Module2002.Output.SkillOutput.SkillOutput14.ParameterOutput.ParameterOutput1 := Module[2].Output.SkillOutput[14].ParameterOutput[1];
Module[2].Input.SkillInput[14].ParameterInput[2] := Module2002.Input.SkillInput.SkillInput14.ParameterInput.ParameterInput2;
Module2002.Output.SkillOutput.SkillOutput14.ParameterOutput.ParameterOutput2 := Module[2].Output.SkillOutput[14].ParameterOutput[2];
Module[2].Input.SkillInput[14].ParameterInput[3] := Module2002.Input.SkillInput.SkillInput14.ParameterInput.ParameterInput3;
Module2002.Output.SkillOutput.SkillOutput14.ParameterOutput.ParameterOutput3 := Module[2].Output.SkillOutput[14].ParameterOutput[3];
Module[2].Input.SkillInput[14].ParameterInput[4] := Module2002.Input.SkillInput.SkillInput14.ParameterInput.ParameterInput4;
Module2002.Output.SkillOutput.SkillOutput14.ParameterOutput.ParameterOutput4 := Module[2].Output.SkillOutput[14].ParameterOutput[4];
Module[2].Input.SkillInput[14].ParameterInput[5] := Module2002.Input.SkillInput.SkillInput14.ParameterInput.ParameterInput5;
Module2002.Output.SkillOutput.SkillOutput14.ParameterOutput.ParameterOutput5 := Module[2].Output.SkillOutput[14].ParameterOutput[5];
Module[2].Input.SkillInput[15].Execute := Module2002.Input.SkillInput.SkillInput15.Execute;
Module2002.Output.SkillOutput.SkillOutput15.Dummy := Module[2].Output.SkillOutput[15].Dummy;
Module2002.Output.SkillOutput.SkillOutput15.ID := Module[2].Output.SkillOutput[15].ID;
Module2002.Output.SkillOutput.SkillOutput15.Name := Module[2].Output.SkillOutput[15].Name;
Module2002.Output.SkillOutput.SkillOutput15.Activated := Module[2].Output.SkillOutput[15].Activated;
Module2002.Output.SkillOutput.SkillOutput15.Ready := Module[2].Output.SkillOutput[15].Ready;
Module2002.Output.SkillOutput.SkillOutput15.Busy := Module[2].Output.SkillOutput[15].Busy;
Module2002.Output.SkillOutput.SkillOutput15.Done := Module[2].Output.SkillOutput[15].Done;
Module2002.Output.SkillOutput.SkillOutput15.Error := Module[2].Output.SkillOutput[15].Error;
Module2002.Output.Statevalue.Statevalue0 := Module[2].Output.Statevalue[0];
Module2002.Output.Statevalue.Statevalue1 := Module[2].Output.Statevalue[1];
Module2002.Output.Statevalue.Statevalue2 := Module[2].Output.Statevalue[2];
Module2002.Output.Statevalue.Statevalue3 := Module[2].Output.Statevalue[3];
Module2002.Output.Statevalue.Statevalue4 := Module[2].Output.Statevalue[4];
Module2002.Output.Statevalue.Statevalue5 := Module[2].Output.Statevalue[5];
Module2002.Output.Statevalue.Statevalue6 := Module[2].Output.Statevalue[6];
Module2002.Output.Statevalue.Statevalue7 := Module[2].Output.Statevalue[7];
Module2002.Output.Statevalue.Statevalue8 := Module[2].Output.Statevalue[8];
Module2002.Output.Statevalue.Statevalue9 := Module[2].Output.Statevalue[9];
Module2002.Output.Statevalue.Statevalue10 := Module[2].Output.Statevalue[10];
Module[2].Input.SkillInput[15].ParameterInput[0] := Module2002.Input.SkillInput.SkillInput15.ParameterInput.ParameterInput0;
Module2002.Output.SkillOutput.SkillOutput15.ParameterOutput.ParameterOutput0 := Module[2].Output.SkillOutput[15].ParameterOutput[0];
Module[2].Input.SkillInput[15].ParameterInput[1] := Module2002.Input.SkillInput.SkillInput15.ParameterInput.ParameterInput1;
Module2002.Output.SkillOutput.SkillOutput15.ParameterOutput.ParameterOutput1 := Module[2].Output.SkillOutput[15].ParameterOutput[1];
Module[2].Input.SkillInput[15].ParameterInput[2] := Module2002.Input.SkillInput.SkillInput15.ParameterInput.ParameterInput2;
Module2002.Output.SkillOutput.SkillOutput15.ParameterOutput.ParameterOutput2 := Module[2].Output.SkillOutput[15].ParameterOutput[2];
Module[2].Input.SkillInput[15].ParameterInput[3] := Module2002.Input.SkillInput.SkillInput15.ParameterInput.ParameterInput3;
Module2002.Output.SkillOutput.SkillOutput15.ParameterOutput.ParameterOutput3 := Module[2].Output.SkillOutput[15].ParameterOutput[3];
Module[2].Input.SkillInput[15].ParameterInput[4] := Module2002.Input.SkillInput.SkillInput15.ParameterInput.ParameterInput4;
Module2002.Output.SkillOutput.SkillOutput15.ParameterOutput.ParameterOutput4 := Module[2].Output.SkillOutput[15].ParameterOutput[4];
Module[2].Input.SkillInput[15].ParameterInput[5] := Module2002.Input.SkillInput.SkillInput15.ParameterInput.ParameterInput5;
Module2002.Output.SkillOutput.SkillOutput15.ParameterOutput.ParameterOutput5 := Module[2].Output.SkillOutput[15].ParameterOutput[5];
Module[3].Input.Mode := Module2003.Input.Mode;
Module[3].Input.ConnectionTestInput := Module2003.Input.ConnectionTestInput;
Module[3].Input.PositionInput := Module2003.Input.PositionInput;
Module[3].Input.Watchbit := Module2003.Input.Watchbit;
Module[3].Input.EmergencyStop := Module2003.Input.EmergencyStop;
Module2003.Output.Dummy := Module[3].Output.Dummy;
Module2003.Output.Name := Module[3].Output.Name;
Module2003.Output.ID := Module[3].Output.ID;
Module2003.Output.IP := Module[3].Output.IP;
Module2003.Output.Idle := Module[3].Output.Idle;
Module2003.Output.Connected := Module[3].Output.Connected;
Module2003.Output.Error := Module[3].Output.Error;
Module2003.Output.ErrorID := Module[3].Output.ErrorID;
Module2003.Output.ErrorDescription := Module[3].Output.ErrorDescription;
Module2003.Output.CurrentTaskDescription := Module[3].Output.CurrentTaskDescription;
Module2003.Output.PositionSensor := Module[3].Output.PositionSensor;
Module2003.Output.ConnectionTestOutput := Module[3].Output.ConnectionTestOutput;
Module[3].Input.SkillInput[0].Execute := Module2003.Input.SkillInput.SkillInput0.Execute;
Module2003.Output.SkillOutput.SkillOutput0.Dummy := Module[3].Output.SkillOutput[0].Dummy;
Module2003.Output.SkillOutput.SkillOutput0.ID := Module[3].Output.SkillOutput[0].ID;
Module2003.Output.SkillOutput.SkillOutput0.Name := Module[3].Output.SkillOutput[0].Name;
Module2003.Output.SkillOutput.SkillOutput0.Activated := Module[3].Output.SkillOutput[0].Activated;
Module2003.Output.SkillOutput.SkillOutput0.Ready := Module[3].Output.SkillOutput[0].Ready;
Module2003.Output.SkillOutput.SkillOutput0.Busy := Module[3].Output.SkillOutput[0].Busy;
Module2003.Output.SkillOutput.SkillOutput0.Done := Module[3].Output.SkillOutput[0].Done;
Module2003.Output.SkillOutput.SkillOutput0.Error := Module[3].Output.SkillOutput[0].Error;
Module2003.Output.Statevalue.Statevalue0 := Module[3].Output.Statevalue[0];
Module2003.Output.Statevalue.Statevalue1 := Module[3].Output.Statevalue[1];
Module2003.Output.Statevalue.Statevalue2 := Module[3].Output.Statevalue[2];
Module2003.Output.Statevalue.Statevalue3 := Module[3].Output.Statevalue[3];
Module2003.Output.Statevalue.Statevalue4 := Module[3].Output.Statevalue[4];
Module2003.Output.Statevalue.Statevalue5 := Module[3].Output.Statevalue[5];
Module2003.Output.Statevalue.Statevalue6 := Module[3].Output.Statevalue[6];
Module2003.Output.Statevalue.Statevalue7 := Module[3].Output.Statevalue[7];
Module2003.Output.Statevalue.Statevalue8 := Module[3].Output.Statevalue[8];
Module2003.Output.Statevalue.Statevalue9 := Module[3].Output.Statevalue[9];
Module2003.Output.Statevalue.Statevalue10 := Module[3].Output.Statevalue[10];
Module[3].Input.SkillInput[0].ParameterInput[0] := Module2003.Input.SkillInput.SkillInput0.ParameterInput.ParameterInput0;
Module2003.Output.SkillOutput.SkillOutput0.ParameterOutput.ParameterOutput0 := Module[3].Output.SkillOutput[0].ParameterOutput[0];
Module[3].Input.SkillInput[0].ParameterInput[1] := Module2003.Input.SkillInput.SkillInput0.ParameterInput.ParameterInput1;
Module2003.Output.SkillOutput.SkillOutput0.ParameterOutput.ParameterOutput1 := Module[3].Output.SkillOutput[0].ParameterOutput[1];
Module[3].Input.SkillInput[0].ParameterInput[2] := Module2003.Input.SkillInput.SkillInput0.ParameterInput.ParameterInput2;
Module2003.Output.SkillOutput.SkillOutput0.ParameterOutput.ParameterOutput2 := Module[3].Output.SkillOutput[0].ParameterOutput[2];
Module[3].Input.SkillInput[0].ParameterInput[3] := Module2003.Input.SkillInput.SkillInput0.ParameterInput.ParameterInput3;
Module2003.Output.SkillOutput.SkillOutput0.ParameterOutput.ParameterOutput3 := Module[3].Output.SkillOutput[0].ParameterOutput[3];
Module[3].Input.SkillInput[0].ParameterInput[4] := Module2003.Input.SkillInput.SkillInput0.ParameterInput.ParameterInput4;
Module2003.Output.SkillOutput.SkillOutput0.ParameterOutput.ParameterOutput4 := Module[3].Output.SkillOutput[0].ParameterOutput[4];
Module[3].Input.SkillInput[0].ParameterInput[5] := Module2003.Input.SkillInput.SkillInput0.ParameterInput.ParameterInput5;
Module2003.Output.SkillOutput.SkillOutput0.ParameterOutput.ParameterOutput5 := Module[3].Output.SkillOutput[0].ParameterOutput[5];
Module[3].Input.SkillInput[1].Execute := Module2003.Input.SkillInput.SkillInput1.Execute;
Module2003.Output.SkillOutput.SkillOutput1.Dummy := Module[3].Output.SkillOutput[1].Dummy;
Module2003.Output.SkillOutput.SkillOutput1.ID := Module[3].Output.SkillOutput[1].ID;
Module2003.Output.SkillOutput.SkillOutput1.Name := Module[3].Output.SkillOutput[1].Name;
Module2003.Output.SkillOutput.SkillOutput1.Activated := Module[3].Output.SkillOutput[1].Activated;
Module2003.Output.SkillOutput.SkillOutput1.Ready := Module[3].Output.SkillOutput[1].Ready;
Module2003.Output.SkillOutput.SkillOutput1.Busy := Module[3].Output.SkillOutput[1].Busy;
Module2003.Output.SkillOutput.SkillOutput1.Done := Module[3].Output.SkillOutput[1].Done;
Module2003.Output.SkillOutput.SkillOutput1.Error := Module[3].Output.SkillOutput[1].Error;
Module2003.Output.Statevalue.Statevalue0 := Module[3].Output.Statevalue[0];
Module2003.Output.Statevalue.Statevalue1 := Module[3].Output.Statevalue[1];
Module2003.Output.Statevalue.Statevalue2 := Module[3].Output.Statevalue[2];
Module2003.Output.Statevalue.Statevalue3 := Module[3].Output.Statevalue[3];
Module2003.Output.Statevalue.Statevalue4 := Module[3].Output.Statevalue[4];
Module2003.Output.Statevalue.Statevalue5 := Module[3].Output.Statevalue[5];
Module2003.Output.Statevalue.Statevalue6 := Module[3].Output.Statevalue[6];
Module2003.Output.Statevalue.Statevalue7 := Module[3].Output.Statevalue[7];
Module2003.Output.Statevalue.Statevalue8 := Module[3].Output.Statevalue[8];
Module2003.Output.Statevalue.Statevalue9 := Module[3].Output.Statevalue[9];
Module2003.Output.Statevalue.Statevalue10 := Module[3].Output.Statevalue[10];
Module[3].Input.SkillInput[1].ParameterInput[0] := Module2003.Input.SkillInput.SkillInput1.ParameterInput.ParameterInput0;
Module2003.Output.SkillOutput.SkillOutput1.ParameterOutput.ParameterOutput0 := Module[3].Output.SkillOutput[1].ParameterOutput[0];
Module[3].Input.SkillInput[1].ParameterInput[1] := Module2003.Input.SkillInput.SkillInput1.ParameterInput.ParameterInput1;
Module2003.Output.SkillOutput.SkillOutput1.ParameterOutput.ParameterOutput1 := Module[3].Output.SkillOutput[1].ParameterOutput[1];
Module[3].Input.SkillInput[1].ParameterInput[2] := Module2003.Input.SkillInput.SkillInput1.ParameterInput.ParameterInput2;
Module2003.Output.SkillOutput.SkillOutput1.ParameterOutput.ParameterOutput2 := Module[3].Output.SkillOutput[1].ParameterOutput[2];
Module[3].Input.SkillInput[1].ParameterInput[3] := Module2003.Input.SkillInput.SkillInput1.ParameterInput.ParameterInput3;
Module2003.Output.SkillOutput.SkillOutput1.ParameterOutput.ParameterOutput3 := Module[3].Output.SkillOutput[1].ParameterOutput[3];
Module[3].Input.SkillInput[1].ParameterInput[4] := Module2003.Input.SkillInput.SkillInput1.ParameterInput.ParameterInput4;
Module2003.Output.SkillOutput.SkillOutput1.ParameterOutput.ParameterOutput4 := Module[3].Output.SkillOutput[1].ParameterOutput[4];
Module[3].Input.SkillInput[1].ParameterInput[5] := Module2003.Input.SkillInput.SkillInput1.ParameterInput.ParameterInput5;
Module2003.Output.SkillOutput.SkillOutput1.ParameterOutput.ParameterOutput5 := Module[3].Output.SkillOutput[1].ParameterOutput[5];
Module[3].Input.SkillInput[2].Execute := Module2003.Input.SkillInput.SkillInput2.Execute;
Module2003.Output.SkillOutput.SkillOutput2.Dummy := Module[3].Output.SkillOutput[2].Dummy;
Module2003.Output.SkillOutput.SkillOutput2.ID := Module[3].Output.SkillOutput[2].ID;
Module2003.Output.SkillOutput.SkillOutput2.Name := Module[3].Output.SkillOutput[2].Name;
Module2003.Output.SkillOutput.SkillOutput2.Activated := Module[3].Output.SkillOutput[2].Activated;
Module2003.Output.SkillOutput.SkillOutput2.Ready := Module[3].Output.SkillOutput[2].Ready;
Module2003.Output.SkillOutput.SkillOutput2.Busy := Module[3].Output.SkillOutput[2].Busy;
Module2003.Output.SkillOutput.SkillOutput2.Done := Module[3].Output.SkillOutput[2].Done;
Module2003.Output.SkillOutput.SkillOutput2.Error := Module[3].Output.SkillOutput[2].Error;
Module2003.Output.Statevalue.Statevalue0 := Module[3].Output.Statevalue[0];
Module2003.Output.Statevalue.Statevalue1 := Module[3].Output.Statevalue[1];
Module2003.Output.Statevalue.Statevalue2 := Module[3].Output.Statevalue[2];
Module2003.Output.Statevalue.Statevalue3 := Module[3].Output.Statevalue[3];
Module2003.Output.Statevalue.Statevalue4 := Module[3].Output.Statevalue[4];
Module2003.Output.Statevalue.Statevalue5 := Module[3].Output.Statevalue[5];
Module2003.Output.Statevalue.Statevalue6 := Module[3].Output.Statevalue[6];
Module2003.Output.Statevalue.Statevalue7 := Module[3].Output.Statevalue[7];
Module2003.Output.Statevalue.Statevalue8 := Module[3].Output.Statevalue[8];
Module2003.Output.Statevalue.Statevalue9 := Module[3].Output.Statevalue[9];
Module2003.Output.Statevalue.Statevalue10 := Module[3].Output.Statevalue[10];
Module[3].Input.SkillInput[2].ParameterInput[0] := Module2003.Input.SkillInput.SkillInput2.ParameterInput.ParameterInput0;
Module2003.Output.SkillOutput.SkillOutput2.ParameterOutput.ParameterOutput0 := Module[3].Output.SkillOutput[2].ParameterOutput[0];
Module[3].Input.SkillInput[2].ParameterInput[1] := Module2003.Input.SkillInput.SkillInput2.ParameterInput.ParameterInput1;
Module2003.Output.SkillOutput.SkillOutput2.ParameterOutput.ParameterOutput1 := Module[3].Output.SkillOutput[2].ParameterOutput[1];
Module[3].Input.SkillInput[2].ParameterInput[2] := Module2003.Input.SkillInput.SkillInput2.ParameterInput.ParameterInput2;
Module2003.Output.SkillOutput.SkillOutput2.ParameterOutput.ParameterOutput2 := Module[3].Output.SkillOutput[2].ParameterOutput[2];
Module[3].Input.SkillInput[2].ParameterInput[3] := Module2003.Input.SkillInput.SkillInput2.ParameterInput.ParameterInput3;
Module2003.Output.SkillOutput.SkillOutput2.ParameterOutput.ParameterOutput3 := Module[3].Output.SkillOutput[2].ParameterOutput[3];
Module[3].Input.SkillInput[2].ParameterInput[4] := Module2003.Input.SkillInput.SkillInput2.ParameterInput.ParameterInput4;
Module2003.Output.SkillOutput.SkillOutput2.ParameterOutput.ParameterOutput4 := Module[3].Output.SkillOutput[2].ParameterOutput[4];
Module[3].Input.SkillInput[2].ParameterInput[5] := Module2003.Input.SkillInput.SkillInput2.ParameterInput.ParameterInput5;
Module2003.Output.SkillOutput.SkillOutput2.ParameterOutput.ParameterOutput5 := Module[3].Output.SkillOutput[2].ParameterOutput[5];
Module[3].Input.SkillInput[3].Execute := Module2003.Input.SkillInput.SkillInput3.Execute;
Module2003.Output.SkillOutput.SkillOutput3.Dummy := Module[3].Output.SkillOutput[3].Dummy;
Module2003.Output.SkillOutput.SkillOutput3.ID := Module[3].Output.SkillOutput[3].ID;
Module2003.Output.SkillOutput.SkillOutput3.Name := Module[3].Output.SkillOutput[3].Name;
Module2003.Output.SkillOutput.SkillOutput3.Activated := Module[3].Output.SkillOutput[3].Activated;
Module2003.Output.SkillOutput.SkillOutput3.Ready := Module[3].Output.SkillOutput[3].Ready;
Module2003.Output.SkillOutput.SkillOutput3.Busy := Module[3].Output.SkillOutput[3].Busy;
Module2003.Output.SkillOutput.SkillOutput3.Done := Module[3].Output.SkillOutput[3].Done;
Module2003.Output.SkillOutput.SkillOutput3.Error := Module[3].Output.SkillOutput[3].Error;
Module2003.Output.Statevalue.Statevalue0 := Module[3].Output.Statevalue[0];
Module2003.Output.Statevalue.Statevalue1 := Module[3].Output.Statevalue[1];
Module2003.Output.Statevalue.Statevalue2 := Module[3].Output.Statevalue[2];
Module2003.Output.Statevalue.Statevalue3 := Module[3].Output.Statevalue[3];
Module2003.Output.Statevalue.Statevalue4 := Module[3].Output.Statevalue[4];
Module2003.Output.Statevalue.Statevalue5 := Module[3].Output.Statevalue[5];
Module2003.Output.Statevalue.Statevalue6 := Module[3].Output.Statevalue[6];
Module2003.Output.Statevalue.Statevalue7 := Module[3].Output.Statevalue[7];
Module2003.Output.Statevalue.Statevalue8 := Module[3].Output.Statevalue[8];
Module2003.Output.Statevalue.Statevalue9 := Module[3].Output.Statevalue[9];
Module2003.Output.Statevalue.Statevalue10 := Module[3].Output.Statevalue[10];
Module[3].Input.SkillInput[3].ParameterInput[0] := Module2003.Input.SkillInput.SkillInput3.ParameterInput.ParameterInput0;
Module2003.Output.SkillOutput.SkillOutput3.ParameterOutput.ParameterOutput0 := Module[3].Output.SkillOutput[3].ParameterOutput[0];
Module[3].Input.SkillInput[3].ParameterInput[1] := Module2003.Input.SkillInput.SkillInput3.ParameterInput.ParameterInput1;
Module2003.Output.SkillOutput.SkillOutput3.ParameterOutput.ParameterOutput1 := Module[3].Output.SkillOutput[3].ParameterOutput[1];
Module[3].Input.SkillInput[3].ParameterInput[2] := Module2003.Input.SkillInput.SkillInput3.ParameterInput.ParameterInput2;
Module2003.Output.SkillOutput.SkillOutput3.ParameterOutput.ParameterOutput2 := Module[3].Output.SkillOutput[3].ParameterOutput[2];
Module[3].Input.SkillInput[3].ParameterInput[3] := Module2003.Input.SkillInput.SkillInput3.ParameterInput.ParameterInput3;
Module2003.Output.SkillOutput.SkillOutput3.ParameterOutput.ParameterOutput3 := Module[3].Output.SkillOutput[3].ParameterOutput[3];
Module[3].Input.SkillInput[3].ParameterInput[4] := Module2003.Input.SkillInput.SkillInput3.ParameterInput.ParameterInput4;
Module2003.Output.SkillOutput.SkillOutput3.ParameterOutput.ParameterOutput4 := Module[3].Output.SkillOutput[3].ParameterOutput[4];
Module[3].Input.SkillInput[3].ParameterInput[5] := Module2003.Input.SkillInput.SkillInput3.ParameterInput.ParameterInput5;
Module2003.Output.SkillOutput.SkillOutput3.ParameterOutput.ParameterOutput5 := Module[3].Output.SkillOutput[3].ParameterOutput[5];
Module[3].Input.SkillInput[4].Execute := Module2003.Input.SkillInput.SkillInput4.Execute;
Module2003.Output.SkillOutput.SkillOutput4.Dummy := Module[3].Output.SkillOutput[4].Dummy;
Module2003.Output.SkillOutput.SkillOutput4.ID := Module[3].Output.SkillOutput[4].ID;
Module2003.Output.SkillOutput.SkillOutput4.Name := Module[3].Output.SkillOutput[4].Name;
Module2003.Output.SkillOutput.SkillOutput4.Activated := Module[3].Output.SkillOutput[4].Activated;
Module2003.Output.SkillOutput.SkillOutput4.Ready := Module[3].Output.SkillOutput[4].Ready;
Module2003.Output.SkillOutput.SkillOutput4.Busy := Module[3].Output.SkillOutput[4].Busy;
Module2003.Output.SkillOutput.SkillOutput4.Done := Module[3].Output.SkillOutput[4].Done;
Module2003.Output.SkillOutput.SkillOutput4.Error := Module[3].Output.SkillOutput[4].Error;
Module2003.Output.Statevalue.Statevalue0 := Module[3].Output.Statevalue[0];
Module2003.Output.Statevalue.Statevalue1 := Module[3].Output.Statevalue[1];
Module2003.Output.Statevalue.Statevalue2 := Module[3].Output.Statevalue[2];
Module2003.Output.Statevalue.Statevalue3 := Module[3].Output.Statevalue[3];
Module2003.Output.Statevalue.Statevalue4 := Module[3].Output.Statevalue[4];
Module2003.Output.Statevalue.Statevalue5 := Module[3].Output.Statevalue[5];
Module2003.Output.Statevalue.Statevalue6 := Module[3].Output.Statevalue[6];
Module2003.Output.Statevalue.Statevalue7 := Module[3].Output.Statevalue[7];
Module2003.Output.Statevalue.Statevalue8 := Module[3].Output.Statevalue[8];
Module2003.Output.Statevalue.Statevalue9 := Module[3].Output.Statevalue[9];
Module2003.Output.Statevalue.Statevalue10 := Module[3].Output.Statevalue[10];
Module[3].Input.SkillInput[4].ParameterInput[0] := Module2003.Input.SkillInput.SkillInput4.ParameterInput.ParameterInput0;
Module2003.Output.SkillOutput.SkillOutput4.ParameterOutput.ParameterOutput0 := Module[3].Output.SkillOutput[4].ParameterOutput[0];
Module[3].Input.SkillInput[4].ParameterInput[1] := Module2003.Input.SkillInput.SkillInput4.ParameterInput.ParameterInput1;
Module2003.Output.SkillOutput.SkillOutput4.ParameterOutput.ParameterOutput1 := Module[3].Output.SkillOutput[4].ParameterOutput[1];
Module[3].Input.SkillInput[4].ParameterInput[2] := Module2003.Input.SkillInput.SkillInput4.ParameterInput.ParameterInput2;
Module2003.Output.SkillOutput.SkillOutput4.ParameterOutput.ParameterOutput2 := Module[3].Output.SkillOutput[4].ParameterOutput[2];
Module[3].Input.SkillInput[4].ParameterInput[3] := Module2003.Input.SkillInput.SkillInput4.ParameterInput.ParameterInput3;
Module2003.Output.SkillOutput.SkillOutput4.ParameterOutput.ParameterOutput3 := Module[3].Output.SkillOutput[4].ParameterOutput[3];
Module[3].Input.SkillInput[4].ParameterInput[4] := Module2003.Input.SkillInput.SkillInput4.ParameterInput.ParameterInput4;
Module2003.Output.SkillOutput.SkillOutput4.ParameterOutput.ParameterOutput4 := Module[3].Output.SkillOutput[4].ParameterOutput[4];
Module[3].Input.SkillInput[4].ParameterInput[5] := Module2003.Input.SkillInput.SkillInput4.ParameterInput.ParameterInput5;
Module2003.Output.SkillOutput.SkillOutput4.ParameterOutput.ParameterOutput5 := Module[3].Output.SkillOutput[4].ParameterOutput[5];
Module[3].Input.SkillInput[5].Execute := Module2003.Input.SkillInput.SkillInput5.Execute;
Module2003.Output.SkillOutput.SkillOutput5.Dummy := Module[3].Output.SkillOutput[5].Dummy;
Module2003.Output.SkillOutput.SkillOutput5.ID := Module[3].Output.SkillOutput[5].ID;
Module2003.Output.SkillOutput.SkillOutput5.Name := Module[3].Output.SkillOutput[5].Name;
Module2003.Output.SkillOutput.SkillOutput5.Activated := Module[3].Output.SkillOutput[5].Activated;
Module2003.Output.SkillOutput.SkillOutput5.Ready := Module[3].Output.SkillOutput[5].Ready;
Module2003.Output.SkillOutput.SkillOutput5.Busy := Module[3].Output.SkillOutput[5].Busy;
Module2003.Output.SkillOutput.SkillOutput5.Done := Module[3].Output.SkillOutput[5].Done;
Module2003.Output.SkillOutput.SkillOutput5.Error := Module[3].Output.SkillOutput[5].Error;
Module2003.Output.Statevalue.Statevalue0 := Module[3].Output.Statevalue[0];
Module2003.Output.Statevalue.Statevalue1 := Module[3].Output.Statevalue[1];
Module2003.Output.Statevalue.Statevalue2 := Module[3].Output.Statevalue[2];
Module2003.Output.Statevalue.Statevalue3 := Module[3].Output.Statevalue[3];
Module2003.Output.Statevalue.Statevalue4 := Module[3].Output.Statevalue[4];
Module2003.Output.Statevalue.Statevalue5 := Module[3].Output.Statevalue[5];
Module2003.Output.Statevalue.Statevalue6 := Module[3].Output.Statevalue[6];
Module2003.Output.Statevalue.Statevalue7 := Module[3].Output.Statevalue[7];
Module2003.Output.Statevalue.Statevalue8 := Module[3].Output.Statevalue[8];
Module2003.Output.Statevalue.Statevalue9 := Module[3].Output.Statevalue[9];
Module2003.Output.Statevalue.Statevalue10 := Module[3].Output.Statevalue[10];
Module[3].Input.SkillInput[5].ParameterInput[0] := Module2003.Input.SkillInput.SkillInput5.ParameterInput.ParameterInput0;
Module2003.Output.SkillOutput.SkillOutput5.ParameterOutput.ParameterOutput0 := Module[3].Output.SkillOutput[5].ParameterOutput[0];
Module[3].Input.SkillInput[5].ParameterInput[1] := Module2003.Input.SkillInput.SkillInput5.ParameterInput.ParameterInput1;
Module2003.Output.SkillOutput.SkillOutput5.ParameterOutput.ParameterOutput1 := Module[3].Output.SkillOutput[5].ParameterOutput[1];
Module[3].Input.SkillInput[5].ParameterInput[2] := Module2003.Input.SkillInput.SkillInput5.ParameterInput.ParameterInput2;
Module2003.Output.SkillOutput.SkillOutput5.ParameterOutput.ParameterOutput2 := Module[3].Output.SkillOutput[5].ParameterOutput[2];
Module[3].Input.SkillInput[5].ParameterInput[3] := Module2003.Input.SkillInput.SkillInput5.ParameterInput.ParameterInput3;
Module2003.Output.SkillOutput.SkillOutput5.ParameterOutput.ParameterOutput3 := Module[3].Output.SkillOutput[5].ParameterOutput[3];
Module[3].Input.SkillInput[5].ParameterInput[4] := Module2003.Input.SkillInput.SkillInput5.ParameterInput.ParameterInput4;
Module2003.Output.SkillOutput.SkillOutput5.ParameterOutput.ParameterOutput4 := Module[3].Output.SkillOutput[5].ParameterOutput[4];
Module[3].Input.SkillInput[5].ParameterInput[5] := Module2003.Input.SkillInput.SkillInput5.ParameterInput.ParameterInput5;
Module2003.Output.SkillOutput.SkillOutput5.ParameterOutput.ParameterOutput5 := Module[3].Output.SkillOutput[5].ParameterOutput[5];
Module[3].Input.SkillInput[6].Execute := Module2003.Input.SkillInput.SkillInput6.Execute;
Module2003.Output.SkillOutput.SkillOutput6.Dummy := Module[3].Output.SkillOutput[6].Dummy;
Module2003.Output.SkillOutput.SkillOutput6.ID := Module[3].Output.SkillOutput[6].ID;
Module2003.Output.SkillOutput.SkillOutput6.Name := Module[3].Output.SkillOutput[6].Name;
Module2003.Output.SkillOutput.SkillOutput6.Activated := Module[3].Output.SkillOutput[6].Activated;
Module2003.Output.SkillOutput.SkillOutput6.Ready := Module[3].Output.SkillOutput[6].Ready;
Module2003.Output.SkillOutput.SkillOutput6.Busy := Module[3].Output.SkillOutput[6].Busy;
Module2003.Output.SkillOutput.SkillOutput6.Done := Module[3].Output.SkillOutput[6].Done;
Module2003.Output.SkillOutput.SkillOutput6.Error := Module[3].Output.SkillOutput[6].Error;
Module2003.Output.Statevalue.Statevalue0 := Module[3].Output.Statevalue[0];
Module2003.Output.Statevalue.Statevalue1 := Module[3].Output.Statevalue[1];
Module2003.Output.Statevalue.Statevalue2 := Module[3].Output.Statevalue[2];
Module2003.Output.Statevalue.Statevalue3 := Module[3].Output.Statevalue[3];
Module2003.Output.Statevalue.Statevalue4 := Module[3].Output.Statevalue[4];
Module2003.Output.Statevalue.Statevalue5 := Module[3].Output.Statevalue[5];
Module2003.Output.Statevalue.Statevalue6 := Module[3].Output.Statevalue[6];
Module2003.Output.Statevalue.Statevalue7 := Module[3].Output.Statevalue[7];
Module2003.Output.Statevalue.Statevalue8 := Module[3].Output.Statevalue[8];
Module2003.Output.Statevalue.Statevalue9 := Module[3].Output.Statevalue[9];
Module2003.Output.Statevalue.Statevalue10 := Module[3].Output.Statevalue[10];
Module[3].Input.SkillInput[6].ParameterInput[0] := Module2003.Input.SkillInput.SkillInput6.ParameterInput.ParameterInput0;
Module2003.Output.SkillOutput.SkillOutput6.ParameterOutput.ParameterOutput0 := Module[3].Output.SkillOutput[6].ParameterOutput[0];
Module[3].Input.SkillInput[6].ParameterInput[1] := Module2003.Input.SkillInput.SkillInput6.ParameterInput.ParameterInput1;
Module2003.Output.SkillOutput.SkillOutput6.ParameterOutput.ParameterOutput1 := Module[3].Output.SkillOutput[6].ParameterOutput[1];
Module[3].Input.SkillInput[6].ParameterInput[2] := Module2003.Input.SkillInput.SkillInput6.ParameterInput.ParameterInput2;
Module2003.Output.SkillOutput.SkillOutput6.ParameterOutput.ParameterOutput2 := Module[3].Output.SkillOutput[6].ParameterOutput[2];
Module[3].Input.SkillInput[6].ParameterInput[3] := Module2003.Input.SkillInput.SkillInput6.ParameterInput.ParameterInput3;
Module2003.Output.SkillOutput.SkillOutput6.ParameterOutput.ParameterOutput3 := Module[3].Output.SkillOutput[6].ParameterOutput[3];
Module[3].Input.SkillInput[6].ParameterInput[4] := Module2003.Input.SkillInput.SkillInput6.ParameterInput.ParameterInput4;
Module2003.Output.SkillOutput.SkillOutput6.ParameterOutput.ParameterOutput4 := Module[3].Output.SkillOutput[6].ParameterOutput[4];
Module[3].Input.SkillInput[6].ParameterInput[5] := Module2003.Input.SkillInput.SkillInput6.ParameterInput.ParameterInput5;
Module2003.Output.SkillOutput.SkillOutput6.ParameterOutput.ParameterOutput5 := Module[3].Output.SkillOutput[6].ParameterOutput[5];
Module[3].Input.SkillInput[7].Execute := Module2003.Input.SkillInput.SkillInput7.Execute;
Module2003.Output.SkillOutput.SkillOutput7.Dummy := Module[3].Output.SkillOutput[7].Dummy;
Module2003.Output.SkillOutput.SkillOutput7.ID := Module[3].Output.SkillOutput[7].ID;
Module2003.Output.SkillOutput.SkillOutput7.Name := Module[3].Output.SkillOutput[7].Name;
Module2003.Output.SkillOutput.SkillOutput7.Activated := Module[3].Output.SkillOutput[7].Activated;
Module2003.Output.SkillOutput.SkillOutput7.Ready := Module[3].Output.SkillOutput[7].Ready;
Module2003.Output.SkillOutput.SkillOutput7.Busy := Module[3].Output.SkillOutput[7].Busy;
Module2003.Output.SkillOutput.SkillOutput7.Done := Module[3].Output.SkillOutput[7].Done;
Module2003.Output.SkillOutput.SkillOutput7.Error := Module[3].Output.SkillOutput[7].Error;
Module2003.Output.Statevalue.Statevalue0 := Module[3].Output.Statevalue[0];
Module2003.Output.Statevalue.Statevalue1 := Module[3].Output.Statevalue[1];
Module2003.Output.Statevalue.Statevalue2 := Module[3].Output.Statevalue[2];
Module2003.Output.Statevalue.Statevalue3 := Module[3].Output.Statevalue[3];
Module2003.Output.Statevalue.Statevalue4 := Module[3].Output.Statevalue[4];
Module2003.Output.Statevalue.Statevalue5 := Module[3].Output.Statevalue[5];
Module2003.Output.Statevalue.Statevalue6 := Module[3].Output.Statevalue[6];
Module2003.Output.Statevalue.Statevalue7 := Module[3].Output.Statevalue[7];
Module2003.Output.Statevalue.Statevalue8 := Module[3].Output.Statevalue[8];
Module2003.Output.Statevalue.Statevalue9 := Module[3].Output.Statevalue[9];
Module2003.Output.Statevalue.Statevalue10 := Module[3].Output.Statevalue[10];
Module[3].Input.SkillInput[7].ParameterInput[0] := Module2003.Input.SkillInput.SkillInput7.ParameterInput.ParameterInput0;
Module2003.Output.SkillOutput.SkillOutput7.ParameterOutput.ParameterOutput0 := Module[3].Output.SkillOutput[7].ParameterOutput[0];
Module[3].Input.SkillInput[7].ParameterInput[1] := Module2003.Input.SkillInput.SkillInput7.ParameterInput.ParameterInput1;
Module2003.Output.SkillOutput.SkillOutput7.ParameterOutput.ParameterOutput1 := Module[3].Output.SkillOutput[7].ParameterOutput[1];
Module[3].Input.SkillInput[7].ParameterInput[2] := Module2003.Input.SkillInput.SkillInput7.ParameterInput.ParameterInput2;
Module2003.Output.SkillOutput.SkillOutput7.ParameterOutput.ParameterOutput2 := Module[3].Output.SkillOutput[7].ParameterOutput[2];
Module[3].Input.SkillInput[7].ParameterInput[3] := Module2003.Input.SkillInput.SkillInput7.ParameterInput.ParameterInput3;
Module2003.Output.SkillOutput.SkillOutput7.ParameterOutput.ParameterOutput3 := Module[3].Output.SkillOutput[7].ParameterOutput[3];
Module[3].Input.SkillInput[7].ParameterInput[4] := Module2003.Input.SkillInput.SkillInput7.ParameterInput.ParameterInput4;
Module2003.Output.SkillOutput.SkillOutput7.ParameterOutput.ParameterOutput4 := Module[3].Output.SkillOutput[7].ParameterOutput[4];
Module[3].Input.SkillInput[7].ParameterInput[5] := Module2003.Input.SkillInput.SkillInput7.ParameterInput.ParameterInput5;
Module2003.Output.SkillOutput.SkillOutput7.ParameterOutput.ParameterOutput5 := Module[3].Output.SkillOutput[7].ParameterOutput[5];
Module[3].Input.SkillInput[8].Execute := Module2003.Input.SkillInput.SkillInput8.Execute;
Module2003.Output.SkillOutput.SkillOutput8.Dummy := Module[3].Output.SkillOutput[8].Dummy;
Module2003.Output.SkillOutput.SkillOutput8.ID := Module[3].Output.SkillOutput[8].ID;
Module2003.Output.SkillOutput.SkillOutput8.Name := Module[3].Output.SkillOutput[8].Name;
Module2003.Output.SkillOutput.SkillOutput8.Activated := Module[3].Output.SkillOutput[8].Activated;
Module2003.Output.SkillOutput.SkillOutput8.Ready := Module[3].Output.SkillOutput[8].Ready;
Module2003.Output.SkillOutput.SkillOutput8.Busy := Module[3].Output.SkillOutput[8].Busy;
Module2003.Output.SkillOutput.SkillOutput8.Done := Module[3].Output.SkillOutput[8].Done;
Module2003.Output.SkillOutput.SkillOutput8.Error := Module[3].Output.SkillOutput[8].Error;
Module2003.Output.Statevalue.Statevalue0 := Module[3].Output.Statevalue[0];
Module2003.Output.Statevalue.Statevalue1 := Module[3].Output.Statevalue[1];
Module2003.Output.Statevalue.Statevalue2 := Module[3].Output.Statevalue[2];
Module2003.Output.Statevalue.Statevalue3 := Module[3].Output.Statevalue[3];
Module2003.Output.Statevalue.Statevalue4 := Module[3].Output.Statevalue[4];
Module2003.Output.Statevalue.Statevalue5 := Module[3].Output.Statevalue[5];
Module2003.Output.Statevalue.Statevalue6 := Module[3].Output.Statevalue[6];
Module2003.Output.Statevalue.Statevalue7 := Module[3].Output.Statevalue[7];
Module2003.Output.Statevalue.Statevalue8 := Module[3].Output.Statevalue[8];
Module2003.Output.Statevalue.Statevalue9 := Module[3].Output.Statevalue[9];
Module2003.Output.Statevalue.Statevalue10 := Module[3].Output.Statevalue[10];
Module[3].Input.SkillInput[8].ParameterInput[0] := Module2003.Input.SkillInput.SkillInput8.ParameterInput.ParameterInput0;
Module2003.Output.SkillOutput.SkillOutput8.ParameterOutput.ParameterOutput0 := Module[3].Output.SkillOutput[8].ParameterOutput[0];
Module[3].Input.SkillInput[8].ParameterInput[1] := Module2003.Input.SkillInput.SkillInput8.ParameterInput.ParameterInput1;
Module2003.Output.SkillOutput.SkillOutput8.ParameterOutput.ParameterOutput1 := Module[3].Output.SkillOutput[8].ParameterOutput[1];
Module[3].Input.SkillInput[8].ParameterInput[2] := Module2003.Input.SkillInput.SkillInput8.ParameterInput.ParameterInput2;
Module2003.Output.SkillOutput.SkillOutput8.ParameterOutput.ParameterOutput2 := Module[3].Output.SkillOutput[8].ParameterOutput[2];
Module[3].Input.SkillInput[8].ParameterInput[3] := Module2003.Input.SkillInput.SkillInput8.ParameterInput.ParameterInput3;
Module2003.Output.SkillOutput.SkillOutput8.ParameterOutput.ParameterOutput3 := Module[3].Output.SkillOutput[8].ParameterOutput[3];
Module[3].Input.SkillInput[8].ParameterInput[4] := Module2003.Input.SkillInput.SkillInput8.ParameterInput.ParameterInput4;
Module2003.Output.SkillOutput.SkillOutput8.ParameterOutput.ParameterOutput4 := Module[3].Output.SkillOutput[8].ParameterOutput[4];
Module[3].Input.SkillInput[8].ParameterInput[5] := Module2003.Input.SkillInput.SkillInput8.ParameterInput.ParameterInput5;
Module2003.Output.SkillOutput.SkillOutput8.ParameterOutput.ParameterOutput5 := Module[3].Output.SkillOutput[8].ParameterOutput[5];
Module[3].Input.SkillInput[9].Execute := Module2003.Input.SkillInput.SkillInput9.Execute;
Module2003.Output.SkillOutput.SkillOutput9.Dummy := Module[3].Output.SkillOutput[9].Dummy;
Module2003.Output.SkillOutput.SkillOutput9.ID := Module[3].Output.SkillOutput[9].ID;
Module2003.Output.SkillOutput.SkillOutput9.Name := Module[3].Output.SkillOutput[9].Name;
Module2003.Output.SkillOutput.SkillOutput9.Activated := Module[3].Output.SkillOutput[9].Activated;
Module2003.Output.SkillOutput.SkillOutput9.Ready := Module[3].Output.SkillOutput[9].Ready;
Module2003.Output.SkillOutput.SkillOutput9.Busy := Module[3].Output.SkillOutput[9].Busy;
Module2003.Output.SkillOutput.SkillOutput9.Done := Module[3].Output.SkillOutput[9].Done;
Module2003.Output.SkillOutput.SkillOutput9.Error := Module[3].Output.SkillOutput[9].Error;
Module2003.Output.Statevalue.Statevalue0 := Module[3].Output.Statevalue[0];
Module2003.Output.Statevalue.Statevalue1 := Module[3].Output.Statevalue[1];
Module2003.Output.Statevalue.Statevalue2 := Module[3].Output.Statevalue[2];
Module2003.Output.Statevalue.Statevalue3 := Module[3].Output.Statevalue[3];
Module2003.Output.Statevalue.Statevalue4 := Module[3].Output.Statevalue[4];
Module2003.Output.Statevalue.Statevalue5 := Module[3].Output.Statevalue[5];
Module2003.Output.Statevalue.Statevalue6 := Module[3].Output.Statevalue[6];
Module2003.Output.Statevalue.Statevalue7 := Module[3].Output.Statevalue[7];
Module2003.Output.Statevalue.Statevalue8 := Module[3].Output.Statevalue[8];
Module2003.Output.Statevalue.Statevalue9 := Module[3].Output.Statevalue[9];
Module2003.Output.Statevalue.Statevalue10 := Module[3].Output.Statevalue[10];
Module[3].Input.SkillInput[9].ParameterInput[0] := Module2003.Input.SkillInput.SkillInput9.ParameterInput.ParameterInput0;
Module2003.Output.SkillOutput.SkillOutput9.ParameterOutput.ParameterOutput0 := Module[3].Output.SkillOutput[9].ParameterOutput[0];
Module[3].Input.SkillInput[9].ParameterInput[1] := Module2003.Input.SkillInput.SkillInput9.ParameterInput.ParameterInput1;
Module2003.Output.SkillOutput.SkillOutput9.ParameterOutput.ParameterOutput1 := Module[3].Output.SkillOutput[9].ParameterOutput[1];
Module[3].Input.SkillInput[9].ParameterInput[2] := Module2003.Input.SkillInput.SkillInput9.ParameterInput.ParameterInput2;
Module2003.Output.SkillOutput.SkillOutput9.ParameterOutput.ParameterOutput2 := Module[3].Output.SkillOutput[9].ParameterOutput[2];
Module[3].Input.SkillInput[9].ParameterInput[3] := Module2003.Input.SkillInput.SkillInput9.ParameterInput.ParameterInput3;
Module2003.Output.SkillOutput.SkillOutput9.ParameterOutput.ParameterOutput3 := Module[3].Output.SkillOutput[9].ParameterOutput[3];
Module[3].Input.SkillInput[9].ParameterInput[4] := Module2003.Input.SkillInput.SkillInput9.ParameterInput.ParameterInput4;
Module2003.Output.SkillOutput.SkillOutput9.ParameterOutput.ParameterOutput4 := Module[3].Output.SkillOutput[9].ParameterOutput[4];
Module[3].Input.SkillInput[9].ParameterInput[5] := Module2003.Input.SkillInput.SkillInput9.ParameterInput.ParameterInput5;
Module2003.Output.SkillOutput.SkillOutput9.ParameterOutput.ParameterOutput5 := Module[3].Output.SkillOutput[9].ParameterOutput[5];
Module[3].Input.SkillInput[10].Execute := Module2003.Input.SkillInput.SkillInput10.Execute;
Module2003.Output.SkillOutput.SkillOutput10.Dummy := Module[3].Output.SkillOutput[10].Dummy;
Module2003.Output.SkillOutput.SkillOutput10.ID := Module[3].Output.SkillOutput[10].ID;
Module2003.Output.SkillOutput.SkillOutput10.Name := Module[3].Output.SkillOutput[10].Name;
Module2003.Output.SkillOutput.SkillOutput10.Activated := Module[3].Output.SkillOutput[10].Activated;
Module2003.Output.SkillOutput.SkillOutput10.Ready := Module[3].Output.SkillOutput[10].Ready;
Module2003.Output.SkillOutput.SkillOutput10.Busy := Module[3].Output.SkillOutput[10].Busy;
Module2003.Output.SkillOutput.SkillOutput10.Done := Module[3].Output.SkillOutput[10].Done;
Module2003.Output.SkillOutput.SkillOutput10.Error := Module[3].Output.SkillOutput[10].Error;
Module2003.Output.Statevalue.Statevalue0 := Module[3].Output.Statevalue[0];
Module2003.Output.Statevalue.Statevalue1 := Module[3].Output.Statevalue[1];
Module2003.Output.Statevalue.Statevalue2 := Module[3].Output.Statevalue[2];
Module2003.Output.Statevalue.Statevalue3 := Module[3].Output.Statevalue[3];
Module2003.Output.Statevalue.Statevalue4 := Module[3].Output.Statevalue[4];
Module2003.Output.Statevalue.Statevalue5 := Module[3].Output.Statevalue[5];
Module2003.Output.Statevalue.Statevalue6 := Module[3].Output.Statevalue[6];
Module2003.Output.Statevalue.Statevalue7 := Module[3].Output.Statevalue[7];
Module2003.Output.Statevalue.Statevalue8 := Module[3].Output.Statevalue[8];
Module2003.Output.Statevalue.Statevalue9 := Module[3].Output.Statevalue[9];
Module2003.Output.Statevalue.Statevalue10 := Module[3].Output.Statevalue[10];
Module[3].Input.SkillInput[10].ParameterInput[0] := Module2003.Input.SkillInput.SkillInput10.ParameterInput.ParameterInput0;
Module2003.Output.SkillOutput.SkillOutput10.ParameterOutput.ParameterOutput0 := Module[3].Output.SkillOutput[10].ParameterOutput[0];
Module[3].Input.SkillInput[10].ParameterInput[1] := Module2003.Input.SkillInput.SkillInput10.ParameterInput.ParameterInput1;
Module2003.Output.SkillOutput.SkillOutput10.ParameterOutput.ParameterOutput1 := Module[3].Output.SkillOutput[10].ParameterOutput[1];
Module[3].Input.SkillInput[10].ParameterInput[2] := Module2003.Input.SkillInput.SkillInput10.ParameterInput.ParameterInput2;
Module2003.Output.SkillOutput.SkillOutput10.ParameterOutput.ParameterOutput2 := Module[3].Output.SkillOutput[10].ParameterOutput[2];
Module[3].Input.SkillInput[10].ParameterInput[3] := Module2003.Input.SkillInput.SkillInput10.ParameterInput.ParameterInput3;
Module2003.Output.SkillOutput.SkillOutput10.ParameterOutput.ParameterOutput3 := Module[3].Output.SkillOutput[10].ParameterOutput[3];
Module[3].Input.SkillInput[10].ParameterInput[4] := Module2003.Input.SkillInput.SkillInput10.ParameterInput.ParameterInput4;
Module2003.Output.SkillOutput.SkillOutput10.ParameterOutput.ParameterOutput4 := Module[3].Output.SkillOutput[10].ParameterOutput[4];
Module[3].Input.SkillInput[10].ParameterInput[5] := Module2003.Input.SkillInput.SkillInput10.ParameterInput.ParameterInput5;
Module2003.Output.SkillOutput.SkillOutput10.ParameterOutput.ParameterOutput5 := Module[3].Output.SkillOutput[10].ParameterOutput[5];
Module[3].Input.SkillInput[11].Execute := Module2003.Input.SkillInput.SkillInput11.Execute;
Module2003.Output.SkillOutput.SkillOutput11.Dummy := Module[3].Output.SkillOutput[11].Dummy;
Module2003.Output.SkillOutput.SkillOutput11.ID := Module[3].Output.SkillOutput[11].ID;
Module2003.Output.SkillOutput.SkillOutput11.Name := Module[3].Output.SkillOutput[11].Name;
Module2003.Output.SkillOutput.SkillOutput11.Activated := Module[3].Output.SkillOutput[11].Activated;
Module2003.Output.SkillOutput.SkillOutput11.Ready := Module[3].Output.SkillOutput[11].Ready;
Module2003.Output.SkillOutput.SkillOutput11.Busy := Module[3].Output.SkillOutput[11].Busy;
Module2003.Output.SkillOutput.SkillOutput11.Done := Module[3].Output.SkillOutput[11].Done;
Module2003.Output.SkillOutput.SkillOutput11.Error := Module[3].Output.SkillOutput[11].Error;
Module2003.Output.Statevalue.Statevalue0 := Module[3].Output.Statevalue[0];
Module2003.Output.Statevalue.Statevalue1 := Module[3].Output.Statevalue[1];
Module2003.Output.Statevalue.Statevalue2 := Module[3].Output.Statevalue[2];
Module2003.Output.Statevalue.Statevalue3 := Module[3].Output.Statevalue[3];
Module2003.Output.Statevalue.Statevalue4 := Module[3].Output.Statevalue[4];
Module2003.Output.Statevalue.Statevalue5 := Module[3].Output.Statevalue[5];
Module2003.Output.Statevalue.Statevalue6 := Module[3].Output.Statevalue[6];
Module2003.Output.Statevalue.Statevalue7 := Module[3].Output.Statevalue[7];
Module2003.Output.Statevalue.Statevalue8 := Module[3].Output.Statevalue[8];
Module2003.Output.Statevalue.Statevalue9 := Module[3].Output.Statevalue[9];
Module2003.Output.Statevalue.Statevalue10 := Module[3].Output.Statevalue[10];
Module[3].Input.SkillInput[11].ParameterInput[0] := Module2003.Input.SkillInput.SkillInput11.ParameterInput.ParameterInput0;
Module2003.Output.SkillOutput.SkillOutput11.ParameterOutput.ParameterOutput0 := Module[3].Output.SkillOutput[11].ParameterOutput[0];
Module[3].Input.SkillInput[11].ParameterInput[1] := Module2003.Input.SkillInput.SkillInput11.ParameterInput.ParameterInput1;
Module2003.Output.SkillOutput.SkillOutput11.ParameterOutput.ParameterOutput1 := Module[3].Output.SkillOutput[11].ParameterOutput[1];
Module[3].Input.SkillInput[11].ParameterInput[2] := Module2003.Input.SkillInput.SkillInput11.ParameterInput.ParameterInput2;
Module2003.Output.SkillOutput.SkillOutput11.ParameterOutput.ParameterOutput2 := Module[3].Output.SkillOutput[11].ParameterOutput[2];
Module[3].Input.SkillInput[11].ParameterInput[3] := Module2003.Input.SkillInput.SkillInput11.ParameterInput.ParameterInput3;
Module2003.Output.SkillOutput.SkillOutput11.ParameterOutput.ParameterOutput3 := Module[3].Output.SkillOutput[11].ParameterOutput[3];
Module[3].Input.SkillInput[11].ParameterInput[4] := Module2003.Input.SkillInput.SkillInput11.ParameterInput.ParameterInput4;
Module2003.Output.SkillOutput.SkillOutput11.ParameterOutput.ParameterOutput4 := Module[3].Output.SkillOutput[11].ParameterOutput[4];
Module[3].Input.SkillInput[11].ParameterInput[5] := Module2003.Input.SkillInput.SkillInput11.ParameterInput.ParameterInput5;
Module2003.Output.SkillOutput.SkillOutput11.ParameterOutput.ParameterOutput5 := Module[3].Output.SkillOutput[11].ParameterOutput[5];
Module[3].Input.SkillInput[12].Execute := Module2003.Input.SkillInput.SkillInput12.Execute;
Module2003.Output.SkillOutput.SkillOutput12.Dummy := Module[3].Output.SkillOutput[12].Dummy;
Module2003.Output.SkillOutput.SkillOutput12.ID := Module[3].Output.SkillOutput[12].ID;
Module2003.Output.SkillOutput.SkillOutput12.Name := Module[3].Output.SkillOutput[12].Name;
Module2003.Output.SkillOutput.SkillOutput12.Activated := Module[3].Output.SkillOutput[12].Activated;
Module2003.Output.SkillOutput.SkillOutput12.Ready := Module[3].Output.SkillOutput[12].Ready;
Module2003.Output.SkillOutput.SkillOutput12.Busy := Module[3].Output.SkillOutput[12].Busy;
Module2003.Output.SkillOutput.SkillOutput12.Done := Module[3].Output.SkillOutput[12].Done;
Module2003.Output.SkillOutput.SkillOutput12.Error := Module[3].Output.SkillOutput[12].Error;
Module2003.Output.Statevalue.Statevalue0 := Module[3].Output.Statevalue[0];
Module2003.Output.Statevalue.Statevalue1 := Module[3].Output.Statevalue[1];
Module2003.Output.Statevalue.Statevalue2 := Module[3].Output.Statevalue[2];
Module2003.Output.Statevalue.Statevalue3 := Module[3].Output.Statevalue[3];
Module2003.Output.Statevalue.Statevalue4 := Module[3].Output.Statevalue[4];
Module2003.Output.Statevalue.Statevalue5 := Module[3].Output.Statevalue[5];
Module2003.Output.Statevalue.Statevalue6 := Module[3].Output.Statevalue[6];
Module2003.Output.Statevalue.Statevalue7 := Module[3].Output.Statevalue[7];
Module2003.Output.Statevalue.Statevalue8 := Module[3].Output.Statevalue[8];
Module2003.Output.Statevalue.Statevalue9 := Module[3].Output.Statevalue[9];
Module2003.Output.Statevalue.Statevalue10 := Module[3].Output.Statevalue[10];
Module[3].Input.SkillInput[12].ParameterInput[0] := Module2003.Input.SkillInput.SkillInput12.ParameterInput.ParameterInput0;
Module2003.Output.SkillOutput.SkillOutput12.ParameterOutput.ParameterOutput0 := Module[3].Output.SkillOutput[12].ParameterOutput[0];
Module[3].Input.SkillInput[12].ParameterInput[1] := Module2003.Input.SkillInput.SkillInput12.ParameterInput.ParameterInput1;
Module2003.Output.SkillOutput.SkillOutput12.ParameterOutput.ParameterOutput1 := Module[3].Output.SkillOutput[12].ParameterOutput[1];
Module[3].Input.SkillInput[12].ParameterInput[2] := Module2003.Input.SkillInput.SkillInput12.ParameterInput.ParameterInput2;
Module2003.Output.SkillOutput.SkillOutput12.ParameterOutput.ParameterOutput2 := Module[3].Output.SkillOutput[12].ParameterOutput[2];
Module[3].Input.SkillInput[12].ParameterInput[3] := Module2003.Input.SkillInput.SkillInput12.ParameterInput.ParameterInput3;
Module2003.Output.SkillOutput.SkillOutput12.ParameterOutput.ParameterOutput3 := Module[3].Output.SkillOutput[12].ParameterOutput[3];
Module[3].Input.SkillInput[12].ParameterInput[4] := Module2003.Input.SkillInput.SkillInput12.ParameterInput.ParameterInput4;
Module2003.Output.SkillOutput.SkillOutput12.ParameterOutput.ParameterOutput4 := Module[3].Output.SkillOutput[12].ParameterOutput[4];
Module[3].Input.SkillInput[12].ParameterInput[5] := Module2003.Input.SkillInput.SkillInput12.ParameterInput.ParameterInput5;
Module2003.Output.SkillOutput.SkillOutput12.ParameterOutput.ParameterOutput5 := Module[3].Output.SkillOutput[12].ParameterOutput[5];
Module[3].Input.SkillInput[13].Execute := Module2003.Input.SkillInput.SkillInput13.Execute;
Module2003.Output.SkillOutput.SkillOutput13.Dummy := Module[3].Output.SkillOutput[13].Dummy;
Module2003.Output.SkillOutput.SkillOutput13.ID := Module[3].Output.SkillOutput[13].ID;
Module2003.Output.SkillOutput.SkillOutput13.Name := Module[3].Output.SkillOutput[13].Name;
Module2003.Output.SkillOutput.SkillOutput13.Activated := Module[3].Output.SkillOutput[13].Activated;
Module2003.Output.SkillOutput.SkillOutput13.Ready := Module[3].Output.SkillOutput[13].Ready;
Module2003.Output.SkillOutput.SkillOutput13.Busy := Module[3].Output.SkillOutput[13].Busy;
Module2003.Output.SkillOutput.SkillOutput13.Done := Module[3].Output.SkillOutput[13].Done;
Module2003.Output.SkillOutput.SkillOutput13.Error := Module[3].Output.SkillOutput[13].Error;
Module2003.Output.Statevalue.Statevalue0 := Module[3].Output.Statevalue[0];
Module2003.Output.Statevalue.Statevalue1 := Module[3].Output.Statevalue[1];
Module2003.Output.Statevalue.Statevalue2 := Module[3].Output.Statevalue[2];
Module2003.Output.Statevalue.Statevalue3 := Module[3].Output.Statevalue[3];
Module2003.Output.Statevalue.Statevalue4 := Module[3].Output.Statevalue[4];
Module2003.Output.Statevalue.Statevalue5 := Module[3].Output.Statevalue[5];
Module2003.Output.Statevalue.Statevalue6 := Module[3].Output.Statevalue[6];
Module2003.Output.Statevalue.Statevalue7 := Module[3].Output.Statevalue[7];
Module2003.Output.Statevalue.Statevalue8 := Module[3].Output.Statevalue[8];
Module2003.Output.Statevalue.Statevalue9 := Module[3].Output.Statevalue[9];
Module2003.Output.Statevalue.Statevalue10 := Module[3].Output.Statevalue[10];
Module[3].Input.SkillInput[13].ParameterInput[0] := Module2003.Input.SkillInput.SkillInput13.ParameterInput.ParameterInput0;
Module2003.Output.SkillOutput.SkillOutput13.ParameterOutput.ParameterOutput0 := Module[3].Output.SkillOutput[13].ParameterOutput[0];
Module[3].Input.SkillInput[13].ParameterInput[1] := Module2003.Input.SkillInput.SkillInput13.ParameterInput.ParameterInput1;
Module2003.Output.SkillOutput.SkillOutput13.ParameterOutput.ParameterOutput1 := Module[3].Output.SkillOutput[13].ParameterOutput[1];
Module[3].Input.SkillInput[13].ParameterInput[2] := Module2003.Input.SkillInput.SkillInput13.ParameterInput.ParameterInput2;
Module2003.Output.SkillOutput.SkillOutput13.ParameterOutput.ParameterOutput2 := Module[3].Output.SkillOutput[13].ParameterOutput[2];
Module[3].Input.SkillInput[13].ParameterInput[3] := Module2003.Input.SkillInput.SkillInput13.ParameterInput.ParameterInput3;
Module2003.Output.SkillOutput.SkillOutput13.ParameterOutput.ParameterOutput3 := Module[3].Output.SkillOutput[13].ParameterOutput[3];
Module[3].Input.SkillInput[13].ParameterInput[4] := Module2003.Input.SkillInput.SkillInput13.ParameterInput.ParameterInput4;
Module2003.Output.SkillOutput.SkillOutput13.ParameterOutput.ParameterOutput4 := Module[3].Output.SkillOutput[13].ParameterOutput[4];
Module[3].Input.SkillInput[13].ParameterInput[5] := Module2003.Input.SkillInput.SkillInput13.ParameterInput.ParameterInput5;
Module2003.Output.SkillOutput.SkillOutput13.ParameterOutput.ParameterOutput5 := Module[3].Output.SkillOutput[13].ParameterOutput[5];
Module[3].Input.SkillInput[14].Execute := Module2003.Input.SkillInput.SkillInput14.Execute;
Module2003.Output.SkillOutput.SkillOutput14.Dummy := Module[3].Output.SkillOutput[14].Dummy;
Module2003.Output.SkillOutput.SkillOutput14.ID := Module[3].Output.SkillOutput[14].ID;
Module2003.Output.SkillOutput.SkillOutput14.Name := Module[3].Output.SkillOutput[14].Name;
Module2003.Output.SkillOutput.SkillOutput14.Activated := Module[3].Output.SkillOutput[14].Activated;
Module2003.Output.SkillOutput.SkillOutput14.Ready := Module[3].Output.SkillOutput[14].Ready;
Module2003.Output.SkillOutput.SkillOutput14.Busy := Module[3].Output.SkillOutput[14].Busy;
Module2003.Output.SkillOutput.SkillOutput14.Done := Module[3].Output.SkillOutput[14].Done;
Module2003.Output.SkillOutput.SkillOutput14.Error := Module[3].Output.SkillOutput[14].Error;
Module2003.Output.Statevalue.Statevalue0 := Module[3].Output.Statevalue[0];
Module2003.Output.Statevalue.Statevalue1 := Module[3].Output.Statevalue[1];
Module2003.Output.Statevalue.Statevalue2 := Module[3].Output.Statevalue[2];
Module2003.Output.Statevalue.Statevalue3 := Module[3].Output.Statevalue[3];
Module2003.Output.Statevalue.Statevalue4 := Module[3].Output.Statevalue[4];
Module2003.Output.Statevalue.Statevalue5 := Module[3].Output.Statevalue[5];
Module2003.Output.Statevalue.Statevalue6 := Module[3].Output.Statevalue[6];
Module2003.Output.Statevalue.Statevalue7 := Module[3].Output.Statevalue[7];
Module2003.Output.Statevalue.Statevalue8 := Module[3].Output.Statevalue[8];
Module2003.Output.Statevalue.Statevalue9 := Module[3].Output.Statevalue[9];
Module2003.Output.Statevalue.Statevalue10 := Module[3].Output.Statevalue[10];
Module[3].Input.SkillInput[14].ParameterInput[0] := Module2003.Input.SkillInput.SkillInput14.ParameterInput.ParameterInput0;
Module2003.Output.SkillOutput.SkillOutput14.ParameterOutput.ParameterOutput0 := Module[3].Output.SkillOutput[14].ParameterOutput[0];
Module[3].Input.SkillInput[14].ParameterInput[1] := Module2003.Input.SkillInput.SkillInput14.ParameterInput.ParameterInput1;
Module2003.Output.SkillOutput.SkillOutput14.ParameterOutput.ParameterOutput1 := Module[3].Output.SkillOutput[14].ParameterOutput[1];
Module[3].Input.SkillInput[14].ParameterInput[2] := Module2003.Input.SkillInput.SkillInput14.ParameterInput.ParameterInput2;
Module2003.Output.SkillOutput.SkillOutput14.ParameterOutput.ParameterOutput2 := Module[3].Output.SkillOutput[14].ParameterOutput[2];
Module[3].Input.SkillInput[14].ParameterInput[3] := Module2003.Input.SkillInput.SkillInput14.ParameterInput.ParameterInput3;
Module2003.Output.SkillOutput.SkillOutput14.ParameterOutput.ParameterOutput3 := Module[3].Output.SkillOutput[14].ParameterOutput[3];
Module[3].Input.SkillInput[14].ParameterInput[4] := Module2003.Input.SkillInput.SkillInput14.ParameterInput.ParameterInput4;
Module2003.Output.SkillOutput.SkillOutput14.ParameterOutput.ParameterOutput4 := Module[3].Output.SkillOutput[14].ParameterOutput[4];
Module[3].Input.SkillInput[14].ParameterInput[5] := Module2003.Input.SkillInput.SkillInput14.ParameterInput.ParameterInput5;
Module2003.Output.SkillOutput.SkillOutput14.ParameterOutput.ParameterOutput5 := Module[3].Output.SkillOutput[14].ParameterOutput[5];
Module[3].Input.SkillInput[15].Execute := Module2003.Input.SkillInput.SkillInput15.Execute;
Module2003.Output.SkillOutput.SkillOutput15.Dummy := Module[3].Output.SkillOutput[15].Dummy;
Module2003.Output.SkillOutput.SkillOutput15.ID := Module[3].Output.SkillOutput[15].ID;
Module2003.Output.SkillOutput.SkillOutput15.Name := Module[3].Output.SkillOutput[15].Name;
Module2003.Output.SkillOutput.SkillOutput15.Activated := Module[3].Output.SkillOutput[15].Activated;
Module2003.Output.SkillOutput.SkillOutput15.Ready := Module[3].Output.SkillOutput[15].Ready;
Module2003.Output.SkillOutput.SkillOutput15.Busy := Module[3].Output.SkillOutput[15].Busy;
Module2003.Output.SkillOutput.SkillOutput15.Done := Module[3].Output.SkillOutput[15].Done;
Module2003.Output.SkillOutput.SkillOutput15.Error := Module[3].Output.SkillOutput[15].Error;
Module2003.Output.Statevalue.Statevalue0 := Module[3].Output.Statevalue[0];
Module2003.Output.Statevalue.Statevalue1 := Module[3].Output.Statevalue[1];
Module2003.Output.Statevalue.Statevalue2 := Module[3].Output.Statevalue[2];
Module2003.Output.Statevalue.Statevalue3 := Module[3].Output.Statevalue[3];
Module2003.Output.Statevalue.Statevalue4 := Module[3].Output.Statevalue[4];
Module2003.Output.Statevalue.Statevalue5 := Module[3].Output.Statevalue[5];
Module2003.Output.Statevalue.Statevalue6 := Module[3].Output.Statevalue[6];
Module2003.Output.Statevalue.Statevalue7 := Module[3].Output.Statevalue[7];
Module2003.Output.Statevalue.Statevalue8 := Module[3].Output.Statevalue[8];
Module2003.Output.Statevalue.Statevalue9 := Module[3].Output.Statevalue[9];
Module2003.Output.Statevalue.Statevalue10 := Module[3].Output.Statevalue[10];
Module[3].Input.SkillInput[15].ParameterInput[0] := Module2003.Input.SkillInput.SkillInput15.ParameterInput.ParameterInput0;
Module2003.Output.SkillOutput.SkillOutput15.ParameterOutput.ParameterOutput0 := Module[3].Output.SkillOutput[15].ParameterOutput[0];
Module[3].Input.SkillInput[15].ParameterInput[1] := Module2003.Input.SkillInput.SkillInput15.ParameterInput.ParameterInput1;
Module2003.Output.SkillOutput.SkillOutput15.ParameterOutput.ParameterOutput1 := Module[3].Output.SkillOutput[15].ParameterOutput[1];
Module[3].Input.SkillInput[15].ParameterInput[2] := Module2003.Input.SkillInput.SkillInput15.ParameterInput.ParameterInput2;
Module2003.Output.SkillOutput.SkillOutput15.ParameterOutput.ParameterOutput2 := Module[3].Output.SkillOutput[15].ParameterOutput[2];
Module[3].Input.SkillInput[15].ParameterInput[3] := Module2003.Input.SkillInput.SkillInput15.ParameterInput.ParameterInput3;
Module2003.Output.SkillOutput.SkillOutput15.ParameterOutput.ParameterOutput3 := Module[3].Output.SkillOutput[15].ParameterOutput[3];
Module[3].Input.SkillInput[15].ParameterInput[4] := Module2003.Input.SkillInput.SkillInput15.ParameterInput.ParameterInput4;
Module2003.Output.SkillOutput.SkillOutput15.ParameterOutput.ParameterOutput4 := Module[3].Output.SkillOutput[15].ParameterOutput[4];
Module[3].Input.SkillInput[15].ParameterInput[5] := Module2003.Input.SkillInput.SkillInput15.ParameterInput.ParameterInput5;
Module2003.Output.SkillOutput.SkillOutput15.ParameterOutput.ParameterOutput5 := Module[3].Output.SkillOutput[15].ParameterOutput[5];
END_IF

END_FUNCTION_BLOCK

(* stored: Version 1.1.0.1, ProductVersion 3.1.0.25
   POU FB_TranslateInterface: Id {c87b2e64-48ac-4f44-bd38-bd248b0423d0} *)
